Universal Robots PolyScope program: main.urp

ProgramRoot directory=/programs/ropax; kinematics=(a=[0, -0.612, -0.5723, 0, 0, 0], d=[0.1273, 0, 0, 0.16394, 0.1157, 0.0922], alpha=[1.5708, 0, 0, 1.5708, -1.5708, 0], deltaTheta=[0, 0, 0, 0, 0, 0], status=notInitialized); name=main; programVersion=(project__name=PolyScope, major__version=1, minor__version=8, svn__revision=25319, build__date=Oct 19 2016, 16:34:22); robotEnvironmentFileName=default; serialNumberRobot=2013202566
  MainProgram cartesianAcceleration=1.2; cartesianSpeed=0.25; jointAcceleration=1.3962634015954636; jointSpeed=1.0471975511965976; moveAsFastAsPossible=true; sharedProcessMoveBlendRadius=0.025; featureReference=(installationNameReference=Base); motionType=JOINT_SPACE
    Script type=1; cachedFileContents=textmsg(get_actual_joint_positions())
      | textmsg("-0-0-0-0-0-0-0-0-0-0-0-0")
      | textmsg(get_actual_tcp_pose()); scriptFile=/programs/ropax/main_cycle.urp
